FUNCTION_BLOCK DIN2TIMEs (* Basic Function Block Type *)
  (* Standard: 61499-2 *)
  (* Version 0.0, 5/23/2024, SESA713705, Schneider Electric, Template *)
  PACKAGE SE.Nereda;
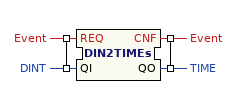
  EVENT_INPUT
    REQ WITH QI; (* Normal Execution Request *)
  END_EVENT
  EVENT_OUTPUT
    CNF WITH QO; (* Execution Confirmation *)
  END_EVENT
  VAR_INPUT
    QI : DINT; (* Input event qualifier *)
  END_VAR
  VAR_OUTPUT
    QO : TIME; (* Output event qualifier *)
  END_VAR
  VAR
    Minutes : REAL;
  END_VAR
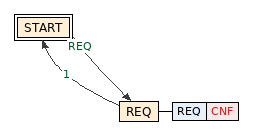
  EC_STATES
    START; (* Initial State *)
    REQ : REQ -> CNF; (* Normal execution *)
  END_STATES
  EC_TRANSITIONS
    START TO REQ := REQ;
    REQ TO START := 1;
  END_TRANSITIONS
  ALGORITHM REQ IN ST: (* Normally executed algorithm *)
;

QO := DINT_TO_TIME(QI * 1000);
  END_ALGORITHM
END_FUNCTION_BLOCK
